// TIA Portal V17 export
// export: Created 2021-12-20T22:44:17.7773066Z, ExportSetting WithDefaults, DisplayName Totally Integrated Automation Portal, DisplayVersion V17, DisplayName TIA Portal Openness, DisplayVersion V17, DisplayName TIA Portal Version Control Interface, DisplayVersion V17, DisplayName STEP 7 Professional, DisplayVersion V17, DisplayName STEP 7 Safety, DisplayVersion V17, DisplayName WinCC Professional, DisplayVersion V17
DATA_BLOCK "NodeRed"   // DB1
{ S7_Optimized_Access := 'FALSE' }
VERSION : 0.1
// stored: AutoNumber true, DBAccessibleFromOPCUA true, IsOnlyStoredInLoadMemory false, IsWriteProtectedInAS false
   VAR
      Trigger : Bool;
      Out : Bool;
      Reset : Bool;
      No_Tolva : Int;
      Tiempo_transcurrido_Tolva : Array[0..10] of Struct
         Timer_1_TON_seg : Int;
         Timer_2_TON_seg : Int;
         Timer_1_TOF_seg : Int;
         Timer_2_TOF_seg : Int;
      END_STRUCT;
      Setpoint_seg : Int;
      No_Timer : Int;
   END_VAR
BEGIN
END_DATA_BLOCK
